// TwinCAT 3 PLC project Opslagvat
// ProgramVersion: 3.1.4024.0
// libraries:
//   Tc2_Standard, * (Beckhoff Automation GmbH)
//   Tc2_System, * (Beckhoff Automation GmbH)
//   Tc3_Module, * (Beckhoff Automation GmbH)
// project tree:
//   / PlcTask.TcTTO (not stored)
//   POUs/ MAIN.TcPOU

// ---- POUs/MAIN.TcPOU
PROGRAM MAIN
VAR
	
// Inputs
	SensorHoog AT %I*: BOOL; // Zijwand  niveau Hoog
	SensorLaag AT %I*: BOOL; // Zijwand  niveau Laag
	StartDrukknop AT %I*: BOOL; // Start DK
	StopDrukknop  AT %I*: BOOL;	// Stop DK

// Outputs
	K1 AT %Q*: BOOL; // Klep
	P1 AT %Q*: BOOL; // Pomp
	
END_VAR

(*
Opslagvat (4 regels code)

Een opslagvat heeft twee sensoren in de zijwand die een laag en hoog niveau aanduiden. 
Aan de hand van een PLC programma dient er automatisch de klep bovenaan het vat geopend te worden als het vat leeg is.
De tank wordt nu gevuld. Als de tank vol is sluit de klep K1 eveneens automatisch. 
Onderaan de tank bevindt zich een pomp P1 die met een start- en stop-drukknop in- en uitgeschakeld kan worden. 

Als de tank leeg gelopen is, stopt de pomp automatisch en opent de klep K1 bovenaan. 
De pomp kan niet ingeschakeld worden zolang de tank gevuld wordt.
*)

K1 := NOT SensorLaag OR SensorHoog; // Open/Sluit klep gebaseerd op sensoren
P1 := StartDrukknop AND NOT SensorHoog AND SensorLaag; // Start/Stop pomp gebaseerd op sensoren en drukknoppen
IF StopDrukknop OR NOT SensorLaag THEN P1 := FALSE; END_IF; // Stop pomp met StopDrukknop of als tank leeg is

END_PROGRAM
